TYPE DUT_CS EXTENDS DUT_Control_Base :
STRUCT
	Auto :BOOL;
	Manual :BOOL;
    Interlock :BOOL;
END_STRUCT
END_TYPE

(* stored: Version 1.1.0.1, ProductVersion 3.1.4024.12
   DUT DUT_CS: Id {e732abcf-a155-4995-b42b-f6d81fdc68f6} *)
